FUNCTION_BLOCK EcMasterGetDeviceState IMPLEMENTS IEcTask
VAR_INPUT
END_VAR
VAR_OUTPUT
END_VAR
VAR
	iState : INT;
	getDeviceState : Tc2_EtherCAT.FB_EcGetSlaveState;
	_execute: BOOL;
	_done: BOOL;
	_busy: BOOL;
	_error: BOOL;
	_netId: AMSNETID;
END_VAR

CASE iState OF
	0:
		IF _execute THEN
			_done := FALSE;
			_busy := TRUE;
			_error := FALSE;
			getDeviceState.bExecute := TRUE;
			IF getDeviceState.bBusy THEN
				iState := 10;
				_execute := false;
			END_IF
		END_IF
	10:
		IF NOT getDeviceState.bBusy THEN
			IF NOT getDeviceState.bError THEN
				_done := TRUE;
			ELSE
				_error := TRUE;
			END_IF
			_busy := FALSE;
			getDeviceState.bExecute := FALSE;
			iState := 0;
		END_IF
END_CASE

getDeviceState(sNetId := Tc2_System.F_CreateAmsNetId(nIds := NetId));

{warning 'add method implementation '}
METHOD Abort : BOOL
getDeviceState.bExecute := FALSE;
_busy := FALSE;
_execute := FALSE;
Abort := TRUE;
iState := 0;
END_METHOD

{warning 'add property implementation'}
PROPERTY Busy : BOOL
GET
Busy := _busy;
END_GET
END_PROPERTY

PROPERTY DeviceAddr : uint
GET
DeviceAddr := getDeviceState.nSlaveAddr;
END_GET
SET
getDeviceState.nSlaveAddr := DeviceAddr;
END_SET
END_PROPERTY

PROPERTY DeviceState : ST_EcSlaveState
GET
DeviceState := getDeviceState.state;
END_GET
END_PROPERTY

{warning 'add property implementation'}
PROPERTY Done : BOOL
GET
Done := _done;
END_GET
END_PROPERTY

{warning 'add property implementation'}
PROPERTY Error : BOOL
GET
Error := _error;
END_GET
END_PROPERTY

{warning 'add method implementation '}
METHOD Execute : BOOL
IF NOT getDeviceState.bBusy THEN
	Execute := _execute := true;
END_IF
END_METHOD

{warning 'add property implementation'}
PROPERTY NetID : amsnetid
GET
NetID := _netId;
END_GET
SET
_netId := NetID;
END_SET
END_PROPERTY

END_FUNCTION_BLOCK

(* stored: Version 1.1.0.1, ProductVersion 3.1.4024.11
   POU EcMasterGetDeviceState: Id {eb8111c1-9599-4e7f-b4ed-16bb8cb24a7d}, SpecialFunc None
   Method Abort: Id {e104b3b1-2df6-40a8-99e9-99e7c0335a67}
   Property Busy: Id {9edc9133-c76f-4b22-a73f-42dd585a7434}
   Get Get: Id {45a946fa-b27d-43db-8525-9a5e4197e51d}
   Property DeviceAddr: Id {ebc64cd1-a884-4a3e-9139-cba6ef505cc1}
   Get Get: Id {70cea917-ddaf-4901-b455-8d8d961adbf4}
   Set Set: Id {73939878-9677-4412-848f-c97037a099f9}
   Property DeviceState: Id {332878ad-f505-4ccc-bceb-07ee40865d38}
   Get Get: Id {83d15e0b-b8ab-4681-9980-aa0c447b0dd3}
   Property Done: Id {d82fd663-67d7-4e24-8e04-aeab5813ba9a}
   Get Get: Id {931ea171-48c1-47ab-a7ac-bbb62b3f0ba9}
   Property Error: Id {c3c8af8e-c95e-4ba9-b01c-f6f131715e86}
   Get Get: Id {03b1bf46-ea38-480e-a5ed-3b482ed9416b}
   Method Execute: Id {41d1a2c6-4795-4012-ab56-fb81afa2f80c}
   Property NetID: Id {3cc6e5ae-e852-42bb-bdbb-346fc6877638}
   Get Get: Id {253f88af-6db4-4c91-a932-fa3184f66fc9}
   Set Set: Id {1141340e-161f-468c-8ad7-dbfe7742b4c1} *)
